{attribute addProperty BoxType "EL2535-0000-0016"}
{attribute addProperty Id "Digital_input_1BIT10.1251Ready_to_enableBIT10.1255WarningBIT10.1256ErrorBIT10.1257TxPDO_ToggleBIT10.1259"}
{attribute addProperty CRC "539495579"}
{attribute addProperty SizeInBites "16"}
{attribute addProperty SizeInBytes "2"}
TYPE Status_20280C9B :
STRUCT
	{attribute addProperty Name "Digital_input_1"}
	Digital_input_1 : BIT;
	{attribute 'hide'}
	reserve_1_BIT_0 : BIT;
	{attribute 'hide'}
	reserve_1_BIT_1 : BIT;
	{attribute 'hide'}
	reserve_1_BIT_2 : BIT;
	{attribute addProperty Name "Ready_to_enable"}
	Ready_to_enable : BIT;
	{attribute addProperty Name "Warning"}
	Warning : BIT;
	{attribute addProperty Name "Error"}
	Error : BIT;
	{attribute 'hide'}
	reserve_2 : BIT;
	{attribute 'hide'}
	reserve_3_BIT_0 : BIT;
	{attribute 'hide'}
	reserve_3_BIT_1 : BIT;
	{attribute 'hide'}
	reserve_3_BIT_2 : BIT;
	{attribute 'hide'}
	reserve_3_BIT_3 : BIT;
	{attribute 'hide'}
	reserve_3_BIT_4 : BIT;
	{attribute 'hide'}
	reserve_3_BIT_5 : BIT;
	{attribute 'hide'}
	reserve_3_BIT_6 : BIT;
	{attribute addProperty Name "TxPDO_Toggle"}
	TxPDO_Toggle : BIT;
END_STRUCT
END_TYPE

(* stored: Version 1.2.0.0, ProductVersion 3.1.4024.9
   DUT Status_20280C9B: Id {f3a8dbbf-a7b8-4b0d-94b9-dcb7aeae836e} *)
